{attribute 'qualified_only'}
{attribute 'strict'}
TYPE E_BeamParamTyp :
(
	enum_member := 0
);
END_TYPE

(* stored: Version 1.1.0.1, ProductVersion 3.1.4022.6
   DUT E_BeamParamTyp: Id {9d2fb958-5b16-4ae9-886d-b057961d2bd3} *)
